Xinje XDPPro project, PLC1: XDM-32T4 (software 3.7.4b 2021-06-17)

PROGRAM Ladder

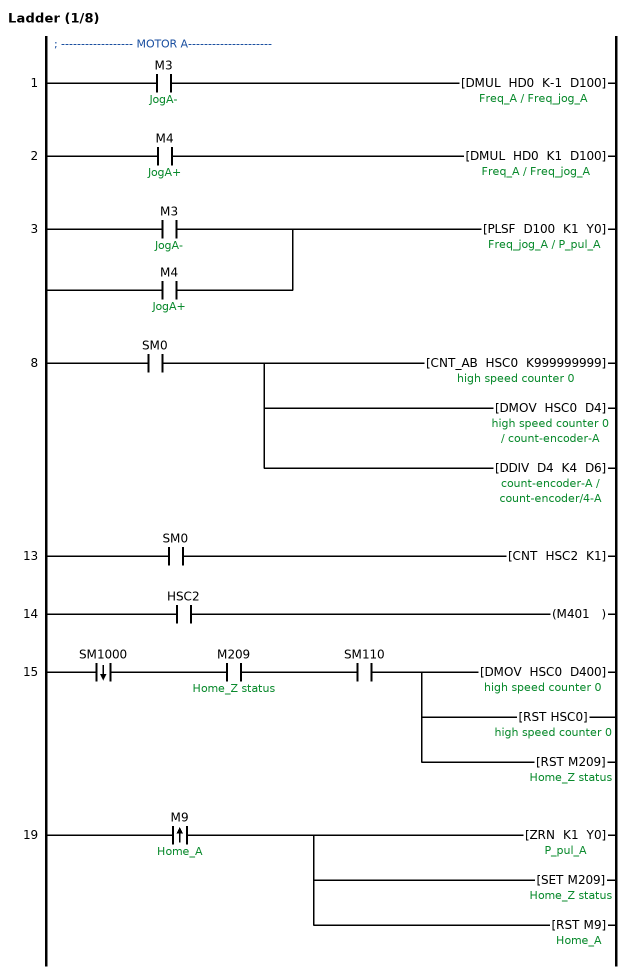
; ------------------ MOTOR A---------------------
LD     M3	; JogA-
DMUL   HD0 K-1 D100	; Freq_A / Freq_jog_A
LD     M4	; JogA+
DMUL   HD0 K1 D100	; Freq_A / Freq_jog_A
LD     M3	; JogA-
OR     M4	; JogA+
PLSF   D100 K1 Y0	; Freq_jog_A / P_pul_A
LD     SM0
CNT_AB HSC0 K999999999	; high speed counter 0
DMOV   HSC0 D4	; high speed counter 0 / count-encoder-A
DDIV   D4 K4 D6	; count-encoder-A / count-encoder/4-A
LD     SM0
CNT    HSC2 K1
LD     HSC2
OUT    M401
LDF    SM1000
AND    M209	; Home_Z status
AND    SM110
DMOV   HSC0 D400	; high speed counter 0
RST    HSC0	; high speed counter 0
RST    M209	; Home_Z status
LDP    M9	; Home_A
ZRN    K1 Y0	; P_pul_A
SET    M209	; Home_Z status
RST    M9	; Home_A

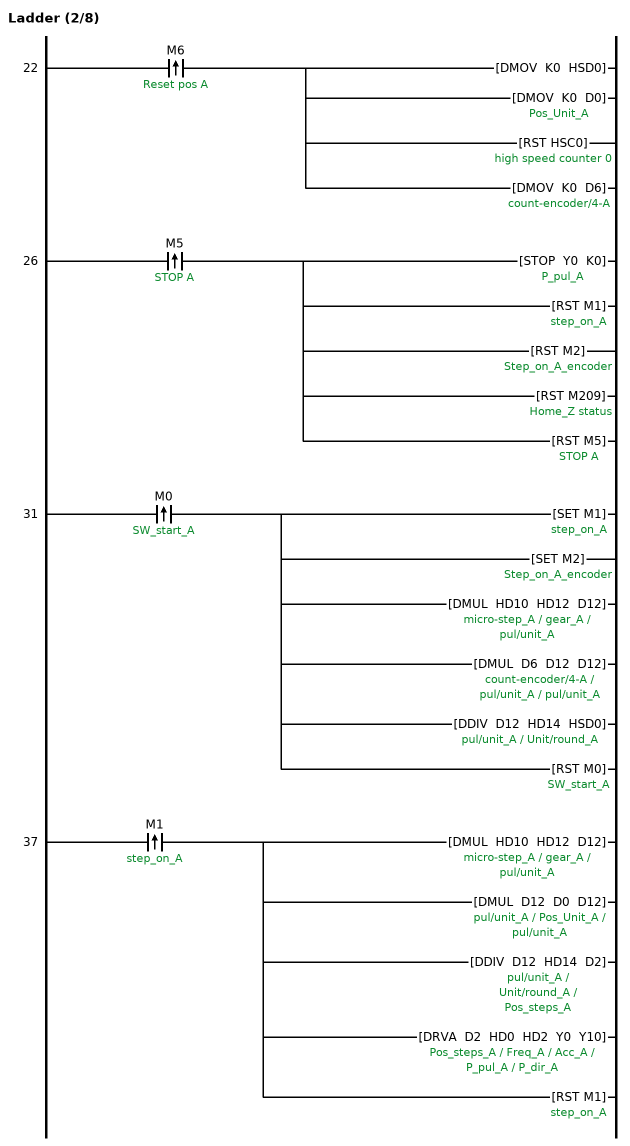
LDP    M6	; Reset pos A
DMOV   K0 HSD0
DMOV   K0 D0	; Pos_Unit_A
RST    HSC0	; high speed counter 0
DMOV   K0 D6	; count-encoder/4-A
LDP    M5	; STOP A
STOP   Y0 K0	; P_pul_A
RST    M1	; step_on_A
RST    M2	; Step_on_A_encoder
RST    M209	; Home_Z status
RST    M5	; STOP A
LDP    M0	; SW_start_A
SET    M1	; step_on_A
SET    M2	; Step_on_A_encoder
DMUL   HD10 HD12 D12	; micro-step_A / gear_A / pul/unit_A
DMUL   D6 D12 D12	; count-encoder/4-A / pul/unit_A / pul/unit_A
DDIV   D12 HD14 HSD0	; pul/unit_A / Unit/round_A
RST    M0	; SW_start_A
LDP    M1	; step_on_A
DMUL   HD10 HD12 D12	; micro-step_A / gear_A / pul/unit_A
DMUL   D12 D0 D12	; pul/unit_A / Pos_Unit_A / pul/unit_A
DDIV   D12 HD14 D2	; pul/unit_A / Unit/round_A / Pos_steps_A
DRVA   D2 HD0 HD2 Y0 Y10	; Pos_steps_A / Freq_A / Acc_A / P_pul_A / P_dir_A
RST    M1	; step_on_A

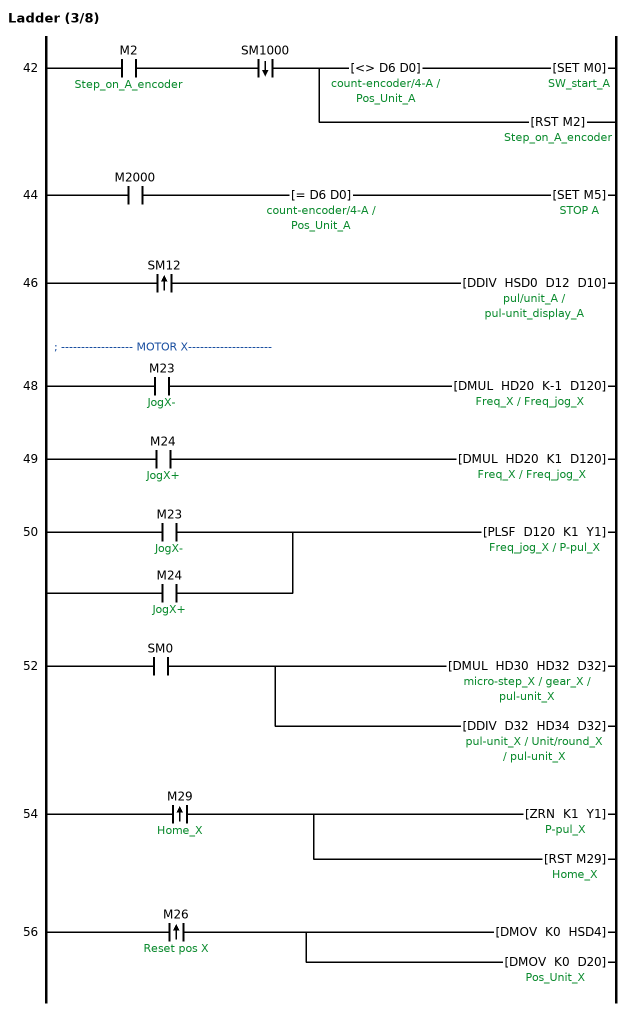
LD     M2	; Step_on_A_encoder
ANDF   SM1000
MPS
AND<>  D6 D0	; count-encoder/4-A / Pos_Unit_A
SET    M0	; SW_start_A
MPP
RST    M2	; Step_on_A_encoder
LD     M2000
AND=   D6 D0	; count-encoder/4-A / Pos_Unit_A
SET    M5	; STOP A
LDP    SM12
DDIV   HSD0 D12 D10	; pul/unit_A / pul-unit_display_A
; ------------------ MOTOR X---------------------
LD     M23	; JogX-
DMUL   HD20 K-1 D120	; Freq_X / Freq_jog_X
LD     M24	; JogX+
DMUL   HD20 K1 D120	; Freq_X / Freq_jog_X
LD     M23	; JogX-
OR     M24	; JogX+
PLSF   D120 K1 Y1	; Freq_jog_X / P-pul_X
LD     SM0
DMUL   HD30 HD32 D32	; micro-step_X / gear_X / pul-unit_X
DDIV   D32 HD34 D32	; pul-unit_X / Unit/round_X / pul-unit_X
LDP    M29	; Home_X
ZRN    K1 Y1	; P-pul_X
RST    M29	; Home_X
LDP    M26	; Reset pos X
DMOV   K0 HSD4
DMOV   K0 D20	; Pos_Unit_X

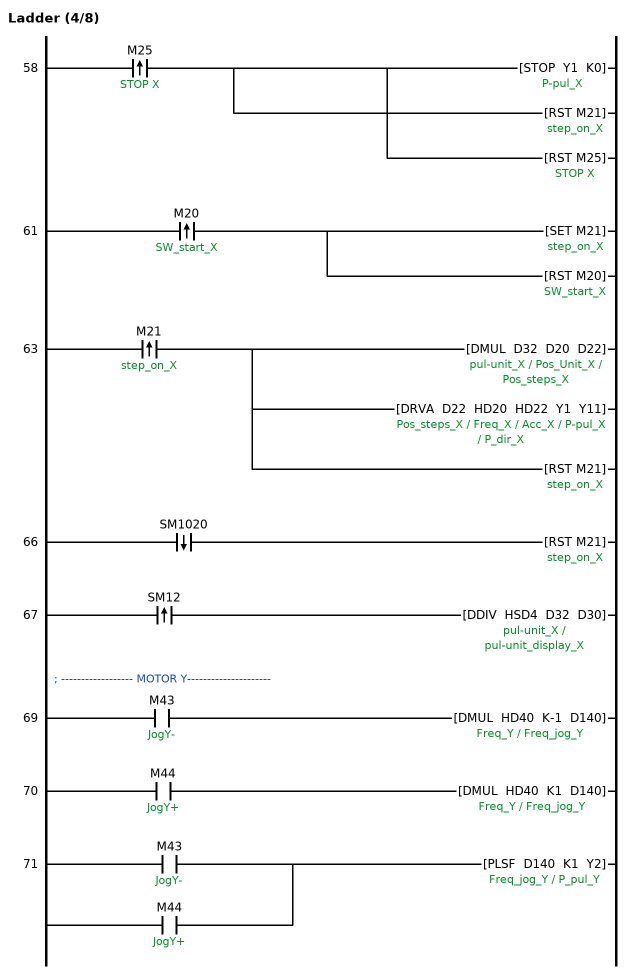
LDP    M25	; STOP X
STOP   Y1 K0	; P-pul_X
RST    M21	; step_on_X
RST    M25	; STOP X
LDP    M20	; SW_start_X
SET    M21	; step_on_X
RST    M20	; SW_start_X
LDP    M21	; step_on_X
DMUL   D32 D20 D22	; pul-unit_X / Pos_Unit_X / Pos_steps_X
DRVA   D22 HD20 HD22 Y1 Y11	; Pos_steps_X / Freq_X / Acc_X / P-pul_X / P_dir_X
RST    M21	; step_on_X
LDF    SM1020
RST    M21	; step_on_X
LDP    SM12
DDIV   HSD4 D32 D30	; pul-unit_X / pul-unit_display_X
; ------------------ MOTOR Y---------------------
LD     M43	; JogY-
DMUL   HD40 K-1 D140	; Freq_Y / Freq_jog_Y
LD     M44	; JogY+
DMUL   HD40 K1 D140	; Freq_Y / Freq_jog_Y
LD     M43	; JogY-
OR     M44	; JogY+
PLSF   D140 K1 Y2	; Freq_jog_Y / P_pul_Y

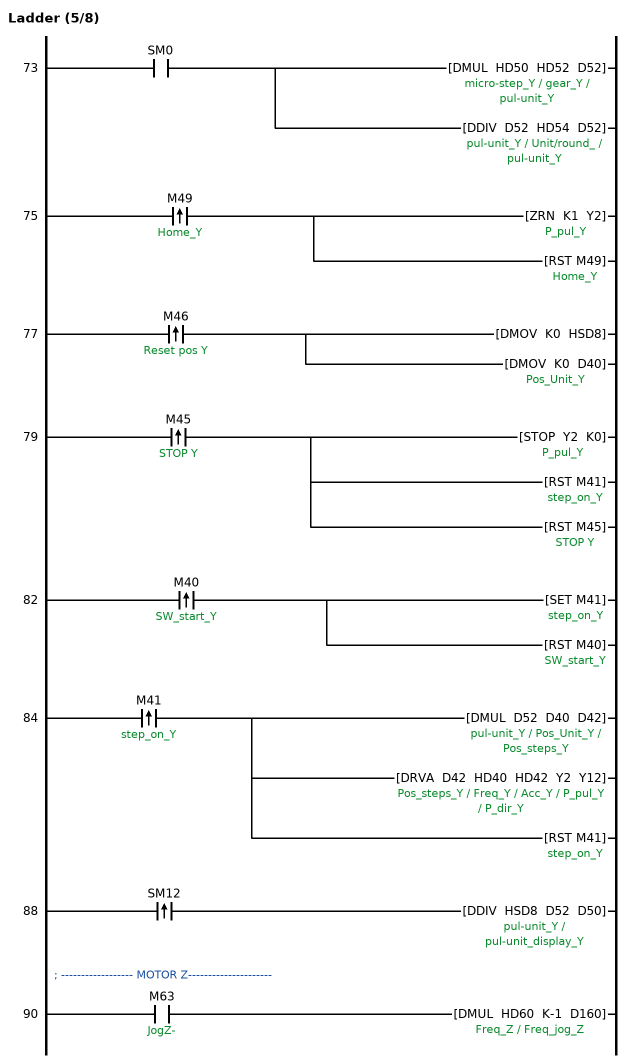
LD     SM0
DMUL   HD50 HD52 D52	; micro-step_Y / gear_Y / pul-unit_Y
DDIV   D52 HD54 D52	; pul-unit_Y / Unit/round_ / pul-unit_Y
LDP    M49	; Home_Y
ZRN    K1 Y2	; P_pul_Y
RST    M49	; Home_Y
LDP    M46	; Reset pos Y
DMOV   K0 HSD8
DMOV   K0 D40	; Pos_Unit_Y
LDP    M45	; STOP Y
STOP   Y2 K0	; P_pul_Y
RST    M41	; step_on_Y
RST    M45	; STOP Y
LDP    M40	; SW_start_Y
SET    M41	; step_on_Y
RST    M40	; SW_start_Y
LDP    M41	; step_on_Y
DMUL   D52 D40 D42	; pul-unit_Y / Pos_Unit_Y / Pos_steps_Y
DRVA   D42 HD40 HD42 Y2 Y12	; Pos_steps_Y / Freq_Y / Acc_Y / P_pul_Y / P_dir_Y
RST    M41	; step_on_Y
LDP    SM12
DDIV   HSD8 D52 D50	; pul-unit_Y / pul-unit_display_Y
; ------------------ MOTOR Z---------------------
LD     M63	; JogZ-
DMUL   HD60 K-1 D160	; Freq_Z / Freq_jog_Z

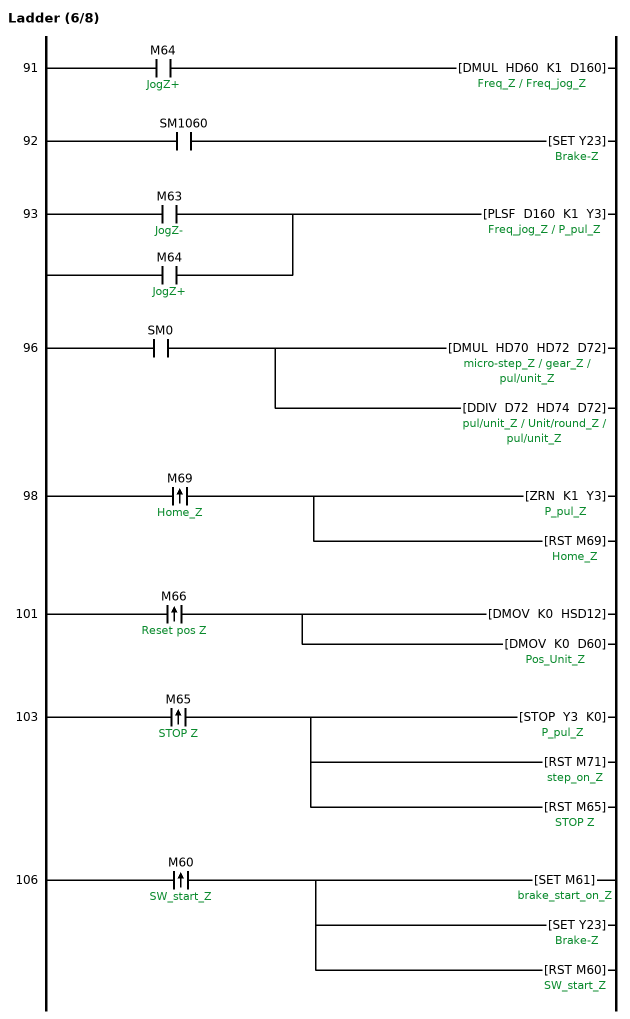
LD     M64	; JogZ+
DMUL   HD60 K1 D160	; Freq_Z / Freq_jog_Z
LD     SM1060
SET    Y23	; Brake-Z
LD     M63	; JogZ-
OR     M64	; JogZ+
PLSF   D160 K1 Y3	; Freq_jog_Z / P_pul_Z
LD     SM0
DMUL   HD70 HD72 D72	; micro-step_Z / gear_Z / pul/unit_Z
DDIV   D72 HD74 D72	; pul/unit_Z / Unit/round_Z / pul/unit_Z
LDP    M69	; Home_Z
ZRN    K1 Y3	; P_pul_Z
RST    M69	; Home_Z
LDP    M66	; Reset pos Z
DMOV   K0 HSD12
DMOV   K0 D60	; Pos_Unit_Z
LDP    M65	; STOP Z
STOP   Y3 K0	; P_pul_Z
RST    M71	; step_on_Z
RST    M65	; STOP Z
LDP    M60	; SW_start_Z
SET    M61	; brake_start_on_Z
SET    Y23	; Brake-Z
RST    M60	; SW_start_Z

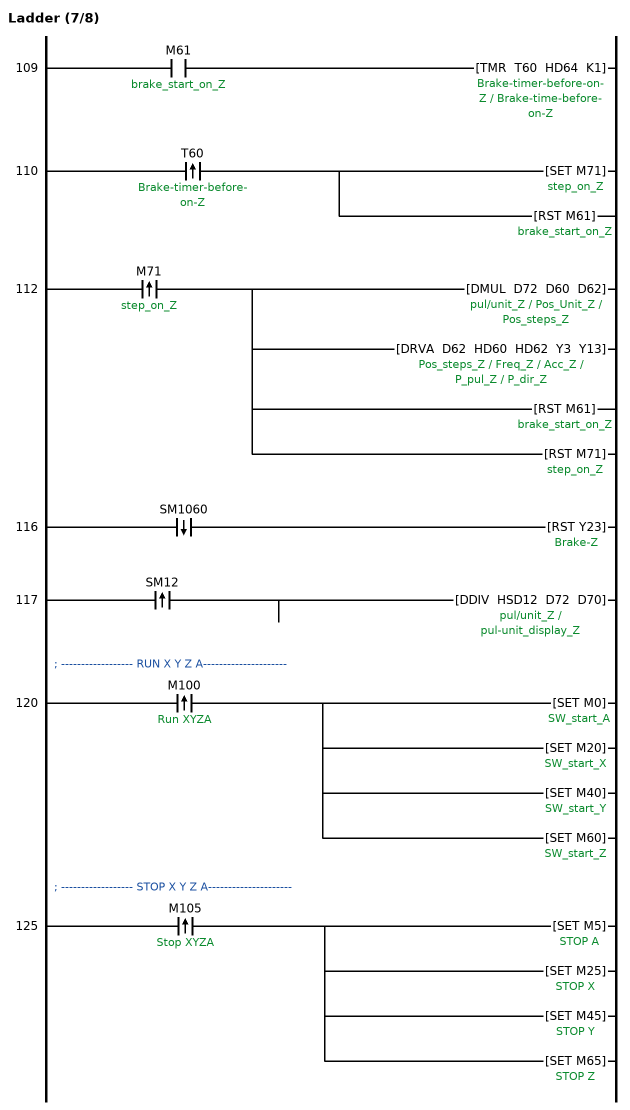
LD     M61	; brake_start_on_Z
TMR    T60 HD64 K1	; Brake-timer-before-on-Z / Brake-time-before-on-Z
LDP    T60	; Brake-timer-before-on-Z
SET    M71	; step_on_Z
RST    M61	; brake_start_on_Z
LDP    M71	; step_on_Z
DMUL   D72 D60 D62	; pul/unit_Z / Pos_Unit_Z / Pos_steps_Z
DRVA   D62 HD60 HD62 Y3 Y13	; Pos_steps_Z / Freq_Z / Acc_Z / P_pul_Z / P_dir_Z
RST    M61	; brake_start_on_Z
RST    M71	; step_on_Z
LDF    SM1060
RST    Y23	; Brake-Z
LDP    SM12
DDIV   HSD12 D72 D70	; pul/unit_Z / pul-unit_display_Z
; ------------------ RUN X Y Z A---------------------
LDP    M100	; Run XYZA
SET    M0	; SW_start_A
SET    M20	; SW_start_X
SET    M40	; SW_start_Y
SET    M60	; SW_start_Z
; ------------------ STOP X Y Z A---------------------
LDP    M105	; Stop XYZA
SET    M5	; STOP A
SET    M25	; STOP X
SET    M45	; STOP Y
SET    M65	; STOP Z

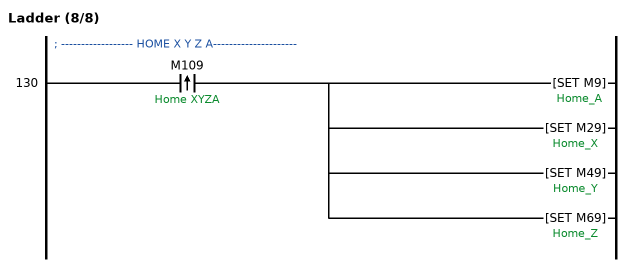
; ------------------ HOME X Y Z A---------------------
LDP    M109	; Home XYZA
SET    M9	; Home_A
SET    M29	; Home_X
SET    M49	; Home_Y
SET    M69	; Home_Z

COMMENTS (devices not used above)
X10	Home-A
X11	Home-X LX-
X12	Home-Y LY-
X13	Home-Z LZ-
M30	Home_flag_X
M50	Home_flag_Y
M70	Home_flag_Z
M10	Home_flag_A
HD4	Pos-encoder-A
HD18	Encoder_x10_A
X21	LX+
X22	LY+
X23	LZ+